// TwinCAT 3 PLC project MudpiSender
// ProgramVersion: 3.1.4023.0
// libraries:
//   ESO ELT Utility Library, * (ESO)
//   ESO LDC Timer Library, * (ESO)
//   Tc2_EtherCAT, * (Beckhoff Automation GmbH)
//   Tc2_Standard, * (Beckhoff Automation GmbH)
//   Tc2_System, * (Beckhoff Automation GmbH)
//   Tc2_Utilities, * (Beckhoff Automation GmbH)
//   Tc3_EventLogger, * (Beckhoff Automation GmbH)
//   Tc3_Module, * (Beckhoff Automation GmbH)
//   VisuDialogs, * (System)
// project tree:
//   DUTs/Structures/ T_PAYLOAD.TcDUT (not stored)
//   / GlobalTextList.TcGTLO (not stored), PlcTask.TcTTO, Visualization Manager.TcVMO (not stored)
//   POUs/ FB_TcExternalTime.TcPOU, MAIN.TcPOU
//   VISUs/ GUI_MUDPI_SENDER.TcVIS, GUI_TIMER.TcVIS (not stored)
// real-time tasks:
//   TASK PlcTask: cycle T#10ms, priority 20, ADS port 350
// I/O:
//   DEVICE Device 1 (RT-Ethernet Adapter)
// variable links:
//   MudpiSender/MudpiSender Instance <-> TcCOM Objects/Object1 (TcNtpExternalTimeProvider)
//     PlcTask Inputs/MAIN.fbTimer.i_exNtpConnected <-> Diagnostic/bIsConnected
//     PlcTask Inputs/MAIN.fbTimer.i_exNtpExtOffset <-> Outputs/nSysToExtTimeOffset
//     PlcTask Inputs/MAIN.fbTimer.i_exNtpExtTime <-> Outputs/nExtTime
//     PlcTask Inputs/MAIN.fbTimer.i_exNtpSynchronized <-> Diagnostic/bIsSynchronized
//     PlcTask Inputs/MAIN.fbTimer.i_exNtpSysTime <-> Outputs/nSysTime

CONFIGURATION MudpiSender
    RESOURCE PLC ON TwinCAT3
        TASK PlcTask(INTERVAL := T#10ms, PRIORITY := 20);
        PROGRAM MAIN WITH PlcTask : MAIN;
    END_RESOURCE
END_CONFIGURATION

// ---- POUs/MAIN.TcPOU
PROGRAM MAIN
VAR
	fbExtTimeSoft : FB_TcExternalTime(ExternalTimeSoft);
	fbSender: FB_MUDPI_SENDER;
	payload: T_PAYLOAD;
	fbTimer: FB_TIME;
	
END_VAR

fbTimer();
fbSender();
payload.data1 := payload.data1 + 1;
fbSender.SetTimestamp(fbTimer.GetMudpiTime());
fbSender.SetMudpiPayload(ADR(payload), SIZEOF(payload));
fbSender.SendData();

END_PROGRAM

// ---- POUs/FB_TcExternalTime.TcPOU
FUNCTION_BLOCK FB_TcExternalTime
VAR
	_hr : HRESULT;
	_ipExtTime : ITcExternalTime;
	_eTimeType: ETcExternalTimeType;
END_VAR

METHOD FB_Exit : BOOL
VAR_INPUT
	bInCopyCode : BOOL; // if TRUE, the exit method is called for exiting an instance that is copied afterwards (online change).
END_VAR
IF _ipExtTime <> 0 THEN
	FW_SafeRelease(ADR(_ipExtTime));
END_IF
END_METHOD

METHOD FB_Init : BOOL
VAR_INPUT
	bInitRetains : BOOL; // if TRUE, the retain variables are initialized (warm start / cold start)
	bInCopyCode : BOOL;  // if TRUE, the instance afterwards gets moved into the copy code (online change)
	eTimeType : ETcExternalTimeType; 
END_VAR
VAR
	ipServer : ITComObjectServer;
END_VAR
ipServer := TwinCAT_SystemInfoVarList._AppInfo.TComSrvPtr;
_eTimeType := eTimeType; 
IF _ipExtTime = 0 THEN
	_hr := ipServer.TcQueryInterface(IID_ITcExternalTime, ADR(_ipExtTime));
	IF FAILED(_hr) THEN RETURN; END_IF
END_IF
END_METHOD

METHOD GetExternalOffset : LINT
VAR_INPUT
END_VAR
IF _ipExtTime <> 0 THEN
	_hr := _ipExtTime.GetExternalTimeOffset(_eTimeType, GetExternalOffset);
	IF _hr <> 0 THEN GetExternalOffset := 0; END_IF
END_IF
END_METHOD

METHOD GetExternalTime : LINT
VAR_INPUT
END_VAR
IF _ipExtTime <> 0 THEN
	GetExternalTime := GetSystemTime();
	_hr := _ipExtTime.SystemTimeToExternalTime(_eTimeType, GetExternalTime);
	IF _hr <> 0 THEN GetExternalTime := 0; END_IF
END_IF
END_METHOD

METHOD GetSystemTime : LINT
GetSystemTime := ULINT_TO_LINT(F_GetSystemTime());
END_METHOD

PROPERTY Result : HRESULT
GET
Result := _hr;
END_GET
END_PROPERTY

END_FUNCTION_BLOCK

// ---- VISUs/GUI_MUDPI_SENDER.TcVIS
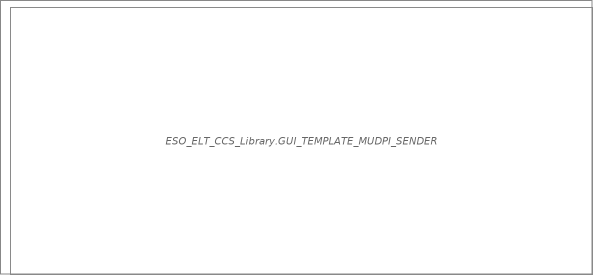
VISUALIZATION GUI_MUDPI_SENDER  // 593x275
    Frame (10,7 583x268)
        shows ESO_ELT_CCS_Library.GUI_TEMPLATE_MUDPI_SENDER(m_Instance := MAIN.fbSender)
END_VISUALIZATION
